// TIA Portal V21 export
VAR_GLOBAL   // PLC tag table "OutputDigitali"
END_VAR
